INTERFACE I_TXTDataExchanger

PROPERTY Active : REFERENCE TO BOOL
GET
END_GET
END_PROPERTY

PROPERTY AmsNetId : STRING
GET
END_GET
SET
END_SET
END_PROPERTY

PROPERTY Busy : REFERENCE TO BOOL
GET
END_GET
END_PROPERTY

PROPERTY Error : REFERENCE TO BOOL
GET
END_GET
END_PROPERTY

PROPERTY ErrorID : REFERENCE TO UDINT
GET
END_GET
END_PROPERTY

PROPERTY FileDir : STRING
GET
END_GET
SET
END_SET
END_PROPERTY

PROPERTY FileName : STRING
GET
END_GET
SET
END_SET
END_PROPERTY

METHOD MR_Abort : BOOL
END_METHOD

METHOD MR_AddMESCommand : BOOL
VAR_INPUT
	sMachineID		: STRING;
	sOperatorID		: STRING;
	sPO				: STRING;
	sProductItem	: STRING;
	bLogOn			: BOOL;
END_VAR
END_METHOD

METHOD MR_Init : BOOL
VAR_INPUT
END_VAR
END_METHOD

METHOD MR_Reset : BOOL
END_METHOD

METHOD MR_SearchForFile : BOOL
VAR_INPUT
	sSearchFileName		: STRING;			(* Whole name of the search file (e.g.: "DemoFile.txt" *)
END_VAR

VAR_OUTPUT
	bFileFound	: BOOL;
END_VAR
END_METHOD

METHOD MR_SelectPath : BOOL
VAR_INPUT
	sFileDir								: STRING; 			(* CSV source file directory name *)
	sFileName 								: STRING; 			(* CSV source file name *)
END_VAR
END_METHOD

PROPERTY Name : STRING
GET
END_GET
SET
END_SET
END_PROPERTY

END_INTERFACE

(* stored: Version 1.1.0.1, ProductVersion 3.1.4024.9
   Itf I_TXTDataExchanger: Id {cc63be76-4c77-41ed-b599-05e5c4d3c908}
   Property Active: Id {916f1107-cd3f-4f75-8f05-839c8d81b7a8}
   Get Get: Id {dfd2e2f0-605f-4528-bd00-e45ae1c21ac9}
   Property AmsNetId: Id {05cbfd4a-3b85-4102-af03-4a7b32e28153}
   Get Get: Id {63786d4a-2018-43bf-a1e9-d7cae1d99042}
   Set Set: Id {7f7dcfa3-93ea-4f47-a75e-dde70b6bd496}
   Property Busy: Id {27c82b83-1da2-46aa-8c10-3e7d98ef3c82}
   Get Get: Id {61a1687e-36a1-4f7e-94d7-c34e5daba583}
   Property Error: Id {4d99b251-f8f9-4c18-b3b7-a0b9370bd389}
   Get Get: Id {8aab9ce4-6ee7-454f-bcd7-43e705483e4a}
   Property ErrorID: Id {350b2ecd-aa25-40f4-8707-3c015f89069f}
   Get Get: Id {a815a143-5b3f-45d1-abf0-86c235a63fe4}
   Property FileDir: Id {65c71048-ddf3-4404-9572-9173ee283968}
   Get Get: Id {b1d3a31d-2dad-4a5d-8f95-9d3b598d5970}
   Set Set: Id {9e2cc943-8b05-4a05-b969-1100212672d4}
   Property FileName: Id {6cfc5e60-1d7f-490b-975c-2a3d4e3a1533}
   Get Get: Id {d660b20d-3e7b-4a59-9fa5-654e7e6b7e03}
   Set Set: Id {9009c8ba-86fd-46a4-90a3-3c2963d14869}
   Method MR_Abort: Id {574d9434-914e-4714-ab26-3e58d53d10f8}
   Method MR_AddMESCommand: Id {f7f1865c-2e00-4351-bac2-1260ec5a7469}
   Method MR_Init: Id {702a7912-0483-4faf-bfc1-cceaae951d77}
   Method MR_Reset: Id {326d4a88-4319-4729-9c74-4946f3a6596f}
   Method MR_SearchForFile: Id {1754118f-214b-4084-b588-46880e96b704}
   Method MR_SelectPath: Id {eb33f0aa-7a55-4a59-aa7b-60b20a5c240a}
   Property Name: Id {d84f5194-8d84-4861-9770-7e986240b630}
   Get Get: Id {01bd6913-86f2-4e4d-b490-cd0bd2813c0b}
   Set Set: Id {1de3d104-9c85-443e-98cc-b4890352627e} *)
